# EPICS substitutions: CARS/iocBoot/iocESP/ESP300.substitutions
file "$(MOTOR)/db/motor.db"
{
pattern
{P,        N,  M,     DTYP,      C,  S,  DESC,       EGU,  DIR,  VELO,  VBAS,  ACCL,  BDST,  BVEL,  BACC,  MRES,  PREC,  DHLM,  DLLM,  INIT}
{ESP300:,  1,  "m1",  "ESP300",  0,  0,  "motor 1",  um,   Pos,  1,     .1,    .2,    0,     1,     .2,    0.01,  5,     100,   -100,  ""}
}
